DATA_BLOCK "DB2017_M_SINA"
TITLE = DB2017_M_SINA
{ S7_Optimized_Access := 'FALSE' }
AUTHOR : ABH
FAMILY : ZeusControl
VERSION : 1.0
//Dispositivo Motor Sinamics
   STRUCT
      M_SINA : Array[0.."N_MAX_DISP_M_SINA"] of "UDT_ZC_DISP_M_SINA";
      Mux { S7_SetPoint := 'False'} : Array[0.."N_MAX_MUX_DISP"] of "UDT_ZC_DISP_MUX_M_SINA";
      Agrup : Array[0.."N_MAX_DISP_AGRUP"] of "UDT_ZC_DISP_AGRUP";
   END_STRUCT;


BEGIN
   M_SINA[0].Hmi_Estado := 0;
   M_SINA[0].Estado_VelocidadLectura := 0.0;
   M_SINA[0].Estado_AutoMan := FALSE;
   M_SINA[0].Estado_Activado := FALSE;
   M_SINA[0].Estado_Enclavado := FALSE;
   M_SINA[0].Estado_PermisoInvertirSentido := FALSE;
   M_SINA[0].Estado_RetornoTermico := FALSE;
   M_SINA[0].Estado_EjeBloqueado := FALSE;
   M_SINA[0].Estado_EjeHabilitado := FALSE;
   M_SINA[0].Alarmas_Termico := FALSE;
   M_SINA[0].Alarmas_SinaSpeed := FALSE;
   M_SINA[0].Alarmas_Mantenimiento := FALSE;
   M_SINA[0].Alarmas_General := FALSE;
   M_SINA[0].Orden_ActivarManual := FALSE;
   M_SINA[0].Orden_ActivarAuto := FALSE;
   M_SINA[0].Orden_ResetHoras := FALSE;
   M_SINA[0].Orden_ResetFallos := FALSE;
   M_SINA[0].Orden_SeleccionInverso := FALSE;
   M_SINA[0].Config_Habilitar := FALSE;
   M_SINA[0].Config_HabilitarRetornoTermico := TRUE;
   M_SINA[0].Config_HabilitarInvertirTermico := TRUE;
   M_SINA[0].Config_HabilitarMantenimiento := FALSE;
   M_SINA[0].Aux_oldActivado := FALSE;
   M_SINA[0].Aux_oldAlarma := FALSE;
   M_SINA[0].Aux_oldAutoMan := FALSE;
   M_SINA[0].Estado_SeguridadOk := TRUE;
   M_SINA[0].Config_GrupoAlarma := 0;
   M_SINA[0].Estado_VelocidadSalida := 0.0;
   M_SINA[0].Estado_Estado := 16#0000;
   M_SINA[0].Estado_CodigoFallo := 16#0000;
   M_SINA[0].Orden_ConsignaManual := 0.0;
   M_SINA[0].Orden_ConsignaAuto := 0.0;
   M_SINA[0].Config_DireccionRetTermicoByte := 0;
   M_SINA[0].Config_DireccionRetTermicoBit := 0;
   M_SINA[0].Config_VelocidadMin := 0.0;
   M_SINA[0].Config_VelocidadMax := 0.0;
   M_SINA[0].Config_K_Velocidad := 50.0;
   M_SINA[0].Tiempos_SetPointTiempoAlarma := 10;
   M_SINA[0].Tiempos_Alarma := 0;
   M_SINA[0].Tiempos_SetPointMantenimiento := 2000.0;
   M_SINA[0].Tiempos_Mantenimiento := 0.0;
   M_SINA[1].Hmi_Estado := 0;
   M_SINA[1].Estado_VelocidadLectura := 0.0;
   M_SINA[1].Estado_AutoMan := FALSE;
   M_SINA[1].Estado_Activado := FALSE;
   M_SINA[1].Estado_Enclavado := FALSE;
   M_SINA[1].Estado_PermisoInvertirSentido := FALSE;
   M_SINA[1].Estado_RetornoTermico := FALSE;
   M_SINA[1].Estado_EjeBloqueado := FALSE;
   M_SINA[1].Estado_EjeHabilitado := FALSE;
   M_SINA[1].Alarmas_Termico := FALSE;
   M_SINA[1].Alarmas_SinaSpeed := FALSE;
   M_SINA[1].Alarmas_Mantenimiento := FALSE;
   M_SINA[1].Alarmas_General := FALSE;
   M_SINA[1].Orden_ActivarManual := FALSE;
   M_SINA[1].Orden_ActivarAuto := FALSE;
   M_SINA[1].Orden_ResetHoras := FALSE;
   M_SINA[1].Orden_ResetFallos := FALSE;
   M_SINA[1].Orden_SeleccionInverso := FALSE;
   M_SINA[1].Config_Habilitar := FALSE;
   M_SINA[1].Config_HabilitarRetornoTermico := TRUE;
   M_SINA[1].Config_HabilitarInvertirTermico := TRUE;
   M_SINA[1].Config_HabilitarMantenimiento := FALSE;
   M_SINA[1].Aux_oldActivado := FALSE;
   M_SINA[1].Aux_oldAlarma := FALSE;
   M_SINA[1].Aux_oldAutoMan := FALSE;
   M_SINA[1].Estado_SeguridadOk := TRUE;
   M_SINA[1].Config_GrupoAlarma := 0;
   M_SINA[1].Estado_VelocidadSalida := 0.0;
   M_SINA[1].Estado_Estado := 16#0000;
   M_SINA[1].Estado_CodigoFallo := 16#0000;
   M_SINA[1].Orden_ConsignaManual := 0.0;
   M_SINA[1].Orden_ConsignaAuto := 0.0;
   M_SINA[1].Config_DireccionRetTermicoByte := 0;
   M_SINA[1].Config_DireccionRetTermicoBit := 0;
   M_SINA[1].Config_VelocidadMin := 0.0;
   M_SINA[1].Config_VelocidadMax := 0.0;
   M_SINA[1].Config_K_Velocidad := 50.0;
   M_SINA[1].Tiempos_SetPointTiempoAlarma := 10;
   M_SINA[1].Tiempos_Alarma := 0;
   M_SINA[1].Tiempos_SetPointMantenimiento := 2000.0;
   M_SINA[1].Tiempos_Mantenimiento := 0.0;
   Mux[0].Habilitar := FALSE;
   Mux[0].ExisteCambio := FALSE;
   Mux[0].MaxVisible := FALSE;
   Mux[0].Index := 0;
   Mux[0].oldIndex := 0;
   Mux[0].M_SINA.Hmi_Estado := 0;
   Mux[0].M_SINA.Estado_VelocidadLectura := 0.0;
   Mux[0].M_SINA.Estado_AutoMan := FALSE;
   Mux[0].M_SINA.Estado_Activado := FALSE;
   Mux[0].M_SINA.Estado_Enclavado := FALSE;
   Mux[0].M_SINA.Estado_PermisoInvertirSentido := FALSE;
   Mux[0].M_SINA.Estado_RetornoTermico := FALSE;
   Mux[0].M_SINA.Estado_EjeBloqueado := FALSE;
   Mux[0].M_SINA.Estado_EjeHabilitado := FALSE;
   Mux[0].M_SINA.Alarmas_Termico := FALSE;
   Mux[0].M_SINA.Alarmas_SinaSpeed := FALSE;
   Mux[0].M_SINA.Alarmas_Mantenimiento := FALSE;
   Mux[0].M_SINA.Alarmas_General := FALSE;
   Mux[0].M_SINA.Orden_ActivarManual := FALSE;
   Mux[0].M_SINA.Orden_ActivarAuto := FALSE;
   Mux[0].M_SINA.Orden_ResetHoras := FALSE;
   Mux[0].M_SINA.Orden_ResetFallos := FALSE;
   Mux[0].M_SINA.Orden_SeleccionInverso := FALSE;
   Mux[0].M_SINA.Config_Habilitar := FALSE;
   Mux[0].M_SINA.Config_HabilitarRetornoTermico := TRUE;
   Mux[0].M_SINA.Config_HabilitarInvertirTermico := TRUE;
   Mux[0].M_SINA.Config_HabilitarMantenimiento := FALSE;
   Mux[0].M_SINA.Aux_oldActivado := FALSE;
   Mux[0].M_SINA.Aux_oldAlarma := FALSE;
   Mux[0].M_SINA.Aux_oldAutoMan := FALSE;
   Mux[0].M_SINA.Estado_SeguridadOk := TRUE;
   Mux[0].M_SINA.Config_GrupoAlarma := 0;
   Mux[0].M_SINA.Estado_VelocidadSalida := 0.0;
   Mux[0].M_SINA.Estado_Estado := 16#0000;
   Mux[0].M_SINA.Estado_CodigoFallo := 16#0000;
   Mux[0].M_SINA.Orden_ConsignaManual := 0.0;
   Mux[0].M_SINA.Orden_ConsignaAuto := 0.0;
   Mux[0].M_SINA.Config_DireccionRetTermicoByte := 0;
   Mux[0].M_SINA.Config_DireccionRetTermicoBit := 0;
   Mux[0].M_SINA.Config_VelocidadMin := 0.0;
   Mux[0].M_SINA.Config_VelocidadMax := 0.0;
   Mux[0].M_SINA.Config_K_Velocidad := 50.0;
   Mux[0].M_SINA.Tiempos_SetPointTiempoAlarma := 10;
   Mux[0].M_SINA.Tiempos_Alarma := 0;
   Mux[0].M_SINA.Tiempos_SetPointMantenimiento := 2000.0;
   Mux[0].M_SINA.Tiempos_Mantenimiento := 0.0;
   Mux[1].Habilitar := FALSE;
   Mux[1].ExisteCambio := FALSE;
   Mux[1].MaxVisible := FALSE;
   Mux[1].Index := 0;
   Mux[1].oldIndex := 0;
   Mux[1].M_SINA.Hmi_Estado := 0;
   Mux[1].M_SINA.Estado_VelocidadLectura := 0.0;
   Mux[1].M_SINA.Estado_AutoMan := FALSE;
   Mux[1].M_SINA.Estado_Activado := FALSE;
   Mux[1].M_SINA.Estado_Enclavado := FALSE;
   Mux[1].M_SINA.Estado_PermisoInvertirSentido := FALSE;
   Mux[1].M_SINA.Estado_RetornoTermico := FALSE;
   Mux[1].M_SINA.Estado_EjeBloqueado := FALSE;
   Mux[1].M_SINA.Estado_EjeHabilitado := FALSE;
   Mux[1].M_SINA.Alarmas_Termico := FALSE;
   Mux[1].M_SINA.Alarmas_SinaSpeed := FALSE;
   Mux[1].M_SINA.Alarmas_Mantenimiento := FALSE;
   Mux[1].M_SINA.Alarmas_General := FALSE;
   Mux[1].M_SINA.Orden_ActivarManual := FALSE;
   Mux[1].M_SINA.Orden_ActivarAuto := FALSE;
   Mux[1].M_SINA.Orden_ResetHoras := FALSE;
   Mux[1].M_SINA.Orden_ResetFallos := FALSE;
   Mux[1].M_SINA.Orden_SeleccionInverso := FALSE;
   Mux[1].M_SINA.Config_Habilitar := FALSE;
   Mux[1].M_SINA.Config_HabilitarRetornoTermico := TRUE;
   Mux[1].M_SINA.Config_HabilitarInvertirTermico := TRUE;
   Mux[1].M_SINA.Config_HabilitarMantenimiento := FALSE;
   Mux[1].M_SINA.Aux_oldActivado := FALSE;
   Mux[1].M_SINA.Aux_oldAlarma := FALSE;
   Mux[1].M_SINA.Aux_oldAutoMan := FALSE;
   Mux[1].M_SINA.Estado_SeguridadOk := TRUE;
   Mux[1].M_SINA.Config_GrupoAlarma := 0;
   Mux[1].M_SINA.Estado_VelocidadSalida := 0.0;
   Mux[1].M_SINA.Estado_Estado := 16#0000;
   Mux[1].M_SINA.Estado_CodigoFallo := 16#0000;
   Mux[1].M_SINA.Orden_ConsignaManual := 0.0;
   Mux[1].M_SINA.Orden_ConsignaAuto := 0.0;
   Mux[1].M_SINA.Config_DireccionRetTermicoByte := 0;
   Mux[1].M_SINA.Config_DireccionRetTermicoBit := 0;
   Mux[1].M_SINA.Config_VelocidadMin := 0.0;
   Mux[1].M_SINA.Config_VelocidadMax := 0.0;
   Mux[1].M_SINA.Config_K_Velocidad := 50.0;
   Mux[1].M_SINA.Tiempos_SetPointTiempoAlarma := 10;
   Mux[1].M_SINA.Tiempos_Alarma := 0;
   Mux[1].M_SINA.Tiempos_SetPointMantenimiento := 2000.0;
   Mux[1].M_SINA.Tiempos_Mantenimiento := 0.0;
   Agrup[0].AlgunaEnManual := TRUE;
   Agrup[0].AlgunaAlarma := FALSE;
   Agrup[0].NuevaAlarma := FALSE;
   Agrup[1].AlgunaEnManual := TRUE;
   Agrup[1].AlgunaAlarma := FALSE;
   Agrup[1].NuevaAlarma := FALSE;

END_DATA_BLOCK

